Fanuc KAREL source: KT00151.KL

PROGRAM KT00151
%NOLOCKGROUP
VAR
  Y1: ARRAY[2] OF BYTE
  H2: ARRAY[2] OF SHORT
  OUT: INTEGER
BEGIN
  Y1[1] = 2
    H2[1] = 3
  OUT = Y1[1] DIV H2[1]
END KT00151
